INTERFACE I_OP_MODE_PAUSE EXTENDS I_OP_MODE

METHOD M_OP_MODE_TO_PAUSE
VAR_INPUT
END_VAR
END_METHOD

PROPERTY P_PAUSE_ACTIVATE : BOOL
GET
END_GET
END_PROPERTY

END_INTERFACE

(* stored: Version 1.1.0.1, ProductVersion 3.1.4024.12
   Itf I_OP_MODE_PAUSE: Id {e1031c58-91ef-4649-aafb-503a551faef1}
   Method M_OP_MODE_TO_PAUSE: Id {f4b2c60b-1b3b-49ea-8b18-dae969926c98}
   Property P_PAUSE_ACTIVATE: Id {4fed84c3-d24e-4583-aa85-6dd88b1dc324}
   Get Get: Id {cc78ba31-4264-4cf0-a39f-1b64704f502e} *)
